FUNCTION_BLOCK PROVIDE_ARR_1024_BYTE (* FB to provide a BYTE array of size 1024 (generic FB) *)
  (* Standard: 61499-2; Description: Copyright (c) 2026 Andreas Demmler Fahrzeugbau This program and the accompanying materials are made available under the terms of the Eclipse Public License 2.0 which is available at https://www.eclipse.org/legal/epl-2.0/ SPDX-License-Identifier: EPL-2.0 This generic Function Block defines an array of 1024 BYTE elements. Functionality: - On the INIT event, the FB reads the array 'D1', calculates its size, and triggers INITO. - The output 'u16DaSize' provides the number of elements in the array. - The 'D1' InOut variable serves as the array container and can be pre-filled with initial values. Example for D1 initialization: [16#01, 16#00, ...] *)
  (* Version 1.1, 2026-03-21, Moritz Ortmeier, Andreas Demmler Fahrzeugbau, changed naming and removed length output *)
  (* Version 1.0, 2026-01-22, Franz H??pfinger, Andreas Demmler Fahrzeugbau *)
  PACKAGE eclipse4diac::convert::providers;
  {SET_ATTRIBUTE(eclipse4diac::core::GenericClassName, 'GEN_INIT_ARR')}
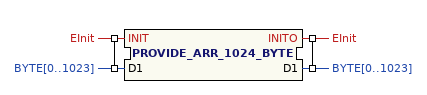
  EVENT_INPUT
    INIT : EInit WITH D1; (* Service Initialization *)
  END_EVENT
  EVENT_OUTPUT
    INITO : EInit WITH D1; (* Initialization Confirm *)
  END_EVENT
  VAR_IN_OUT
    D1 : ARRAY [0..1023] OF BYTE; (* Array in/out *)
  END_VAR
END_FUNCTION_BLOCK
